// TIA Portal V18 export
FUNCTION "DObasic" : Void   // FC10004, FBD
{ S7_Optimized_Access := 'TRUE' }
VERSION : 0.1
// stored: AutoNumber false, IsIECCheckEnabled false, SetENOAutomatically false, UDAEnableTagReadback false
   VAR_INPUT
      xInput : Bool;
      cM0A : Byte;   // 0-direct / 1-reverse / 0-outp_off / 1- aut=1 /2 -out=input
   END_VAR
   VAR_OUTPUT
      iCounter : Int;
      xOutput : Bool;
   END_VAR
   VAR_IN_OUT
      Bit_Count_1 : Bool;
   END_VAR
   VAR_TEMP
      cM0A_0 : Bool;
      cM0A_1 : Bool;
      cM0A_2 : Bool;
   END_VAR
   VAR CONSTANT
      bit_count : Bool;
   END_VAR
   VAR_TEMP   // added for the SCL form of the ladder/FBD networks
      _w1 : Bool;
   END_VAR
BEGIN

REGION Network 1
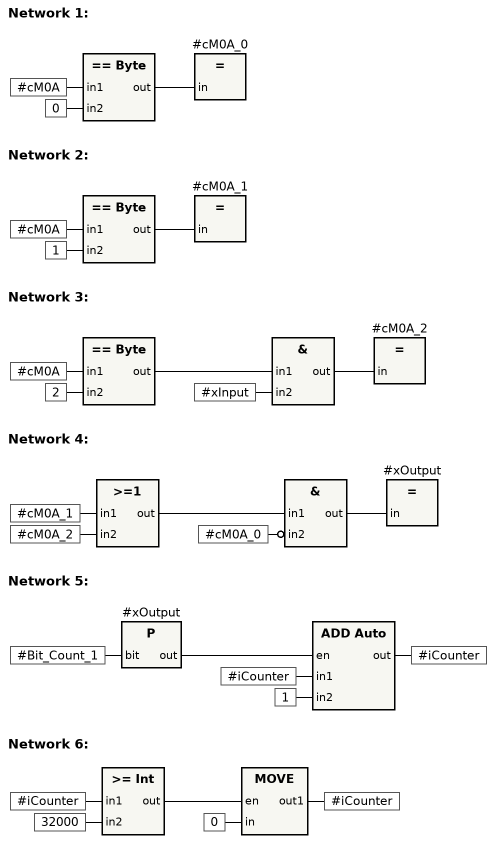
   #cM0A_0 := #cM0A = 0;
END_REGION

REGION Network 2
   #cM0A_1 := #cM0A = 1;
END_REGION

REGION Network 3
   #cM0A_2 := (#cM0A = 2) AND #xInput;
END_REGION

REGION Network 4
   #xOutput := (#cM0A_1 OR #cM0A_2) AND NOT #cM0A_0;
END_REGION

REGION Network 5
   #_w1 := #xOutput AND NOT #Bit_Count_1;   // rising edge of #xOutput
   #Bit_Count_1 := #xOutput;
   IF #_w1 THEN #iCounter := #iCounter + 1; END_IF;
END_REGION

REGION Network 6
   IF #iCounter >= 32000 THEN #iCounter := 0; END_IF;
END_REGION
END_FUNCTION
